// TIA Portal V18 export
DATA_BLOCK "productionCounter_DB"   // DB18
VERSION : 0.1
// stored: AutoNumber true, DBAccessibleFromOPCUA true, DBAccessibleFromWebserver true, InstanceOfName productionCounter, InstanceOfType FB
"productionCounter"
   // VAR_INPUT
   //    I_partProduced : Bool;
   //    I_nokPart : Bool;
   // END_VAR
   // VAR_IN_OUT
   //    IO_actualValues : "UDT_actualValues";
   //    IO_PreviousValues : "UDT_actualValues";
   //    IO_settings : "UDT_settings";
   //    IO_control : "UDT_control";
   //    IO_settingsShift1 : "UDT_settingsShift";
   //    IO_settingsShift2 : "UDT_settingsShift";
   //    IO_settingsShift3 : "UDT_settingsShift";
   //    IO_locTime : DTL;
   // END_VAR
   // VAR
   //    fpBit_resetCounters : Bool;
   //    fpBit_partProduced : Bool;
   //    fpBit_nokPart : Bool;
   //    fpBit_stop : Bool;
   //    fpBit_start : Bool;
   //    RS_taktTimeEn : Bool;
   //    TIM_taktTime { S7_SetPoint := 'True'} : TONR_TIME;
   //    memTaktTime : DInt;
   //    shiftTrigger0 { S7_SetPoint := 'True'} : "shiftTrigger";
   //    shiftTrigger1 { S7_SetPoint := 'True'} : "shiftTrigger";
   //    shiftTrigger2 { S7_SetPoint := 'True'} : "shiftTrigger";
   // END_VAR
BEGIN
END_DATA_BLOCK
